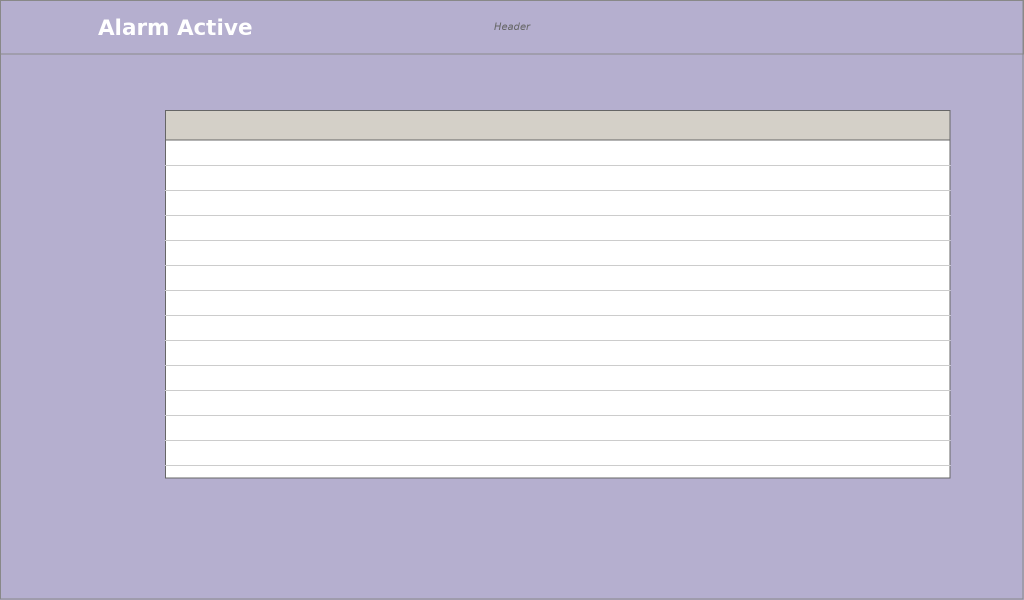
VISUALIZATION AlarmActive  // 1024x600
    Frame (0,-1 1024x55)
        shows Header()
    Label (95,15 250x25), "Alarm Active"
    Table (165,110 785x368), data array: Status_GVL.arAlarmActive
        p3854506369: Status_GVL.arAlarmActive[INDEX].Status
        p1892666644: Status_GVL.arAlarmActive[INDEX].ErrorID
        p338671338: Status_GVL.arAlarmActive[INDEX].ErrorMsg
        p2170511999: Status_GVL.arAlarmActive[INDEX].TimeStop
        p1755163831: Error Message
        p4092479075: Time Stop
END_VISUALIZATION

(* stored: Version 1.1.0.1, ProductVersion 3.1.4024.12
   Visu AlarmActive: Id {898c2db9-7a3a-44d1-b1c1-4776da095824} *)
